// TIA Portal project "QPLC_LADDER" (V16)

(* hardware
DEVICE "S7-1200 station_1"  S7-1200 Station
   slot 0: "Rack_0"  S7-1200 Rack  Rack  V1.0
   slot 1: "PLC_1"  CPU 1214C DC/DC/DC  6ES7 214-1AG40-0XB0  V4.4
   slot 2: "DI 8/DQ 8x24VDC_1"  6ES7 223-1BH32-0XB0  V2.0
*)

// ===== PLC "PLC_1"  CPU 1214C DC/DC/DC =====

VAR_GLOBAL   // PLC tag table "Default tag table"
   "start" AT %I0.0 : Bool;   // Botão começar produção
   "stop" AT %I0.1 : Bool;   // Botão parar produção
   "reset" AT %I0.2 : Bool;   // Botão Reset produção
   "chave" AT %I0.3 : Bool;   // Seleção Modo Automático/Manual
   "Emergência (NO)" AT %I0.4 : Bool;   // Botão de emergencia NO
   "Sen_Peça_Inicial" AT %I0.5 : Bool;   // Sensor detetor de peça
   "Sensor Posição 2" AT %I0.6 : Bool;
   "Sensor Posição 3" AT %I0.7 : Bool;
   "Sen_Gripper_Embaixo" AT %I1.0 : Bool;   // Sensor do braço avançado
   "Sen_Gripper_Em_Cima" AT %I1.1 : Bool;   // Sensor do braço Recuado
   "Sen_Garra_Função" AT %I1.2 : Bool;   // Posição da garra
   "Sensor Posição 1" AT %I1.3 : Bool;   // Posição 1 do braço
   "Prato_Rec" AT %I1.4 : Bool;
   "Prato_Avanc" AT %I1.5 : Bool;
   "Btn_NC_Em" AT %I1.6 : Bool;   // Botão de emergencia NO
   "Pressostato" AT %I1.7 : Bool;
   "LedStart_KA1" AT %Q0.0 : Bool;
   "LedReset_KA2" AT %Q0.1 : Bool;
   "LedQ1_KA3" AT %Q0.2 : Bool;   // Também vai para a o sinalizador da torre
   "LEDQ2_KA4" AT %Q0.3 : Bool;
   "Braço_Direita" AT %Q0.4 : Bool;   // Ordem mover braço para esquerda
   "Braço_Esquerda" AT %Q0.5 : Bool;   // Ordem mover braço para direita
   "Braço_Ação" AT %Q0.6 : Bool;   // Ordem de avanço do braço
   "Garra_AbertaKA8" AT %Q0.7 : Bool;   // Ordem abertura da garra
   "Prato_Rec_KA9" AT %Q1.0 : Bool;   // Ordem recuar o prato
   "Prato_Avan_KA10" AT %Q1.1 : Bool;   // Ordem avançar o prato
   "Valv_KA11" AT %Q1.2 : Bool;
   "System_Byte" AT %MB1 : Byte;
   "FirstScan" AT %M1.0 : Bool;
   "DiagStatusUpdate" AT %M1.1 : Bool;
   "AlwaysTRUE" AT %M1.2 : Bool;
   "AlwaysFALSE" AT %M1.3 : Bool;
   "E_1" AT %M2.0 : Bool;
   "E_2" AT %M2.1 : Bool;
   "E_3" AT %M2.2 : Bool;
   "E_4" AT %M2.3 : Bool;
   "E_5" AT %M2.4 : Bool;
END_VAR

// folder: System blocks/Program resources

DATA_BLOCK "Cooldown para Direita"   // DB1
{ S7_Optimized_Access := 'TRUE' }
AUTHOR : Simatic
FAMILY : IEC
NAME : IEC_TMR
VERSION : 1.0
// stored: InstanceOfName IEC_TIMER
"IEC_TIMER"
BEGIN
END_DATA_BLOCK

DATA_BLOCK "Bit_ON_E2"   // DB2
{ S7_Optimized_Access := 'TRUE' }
AUTHOR : Simatic
FAMILY : IEC
NAME : IEC_TMR
VERSION : 1.0
// stored: InstanceOfName IEC_TIMER
"IEC_TIMER"
BEGIN
END_DATA_BLOCK

// folder: (top level)

FUNCTION "Geral" : Void   // FC1, LAD
{ S7_Optimized_Access := 'TRUE' }
VERSION : 0.1
BEGIN

REGION Network 1: Ordem mover braço para esquerda
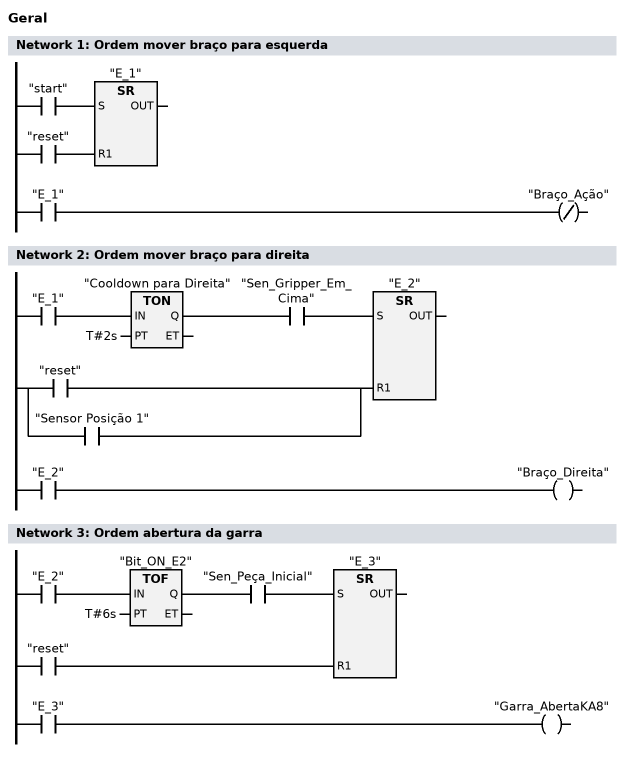
   RUNG wire#powerrail
      Contact( "start" )
      S_SR(operand := "E_1", r1 := wire#w1)
   END_RUNG
   RUNG wire#powerrail
      Contact( "reset" )
   END_RUNG wire#w1
   RUNG wire#powerrail
      Contact( "E_1" )
      I_Coil( "Braço_Ação" )
   END_RUNG
   // the same network as SCL:
   IF "start" THEN
       "E_1" := TRUE;   // SR flip-flop
   END_IF;
   IF "reset" THEN "E_1" := FALSE; END_IF;
   "Braço_Ação" := NOT "E_1";
END_REGION

REGION Network 2: Ordem mover braço para direita
   "Cooldown para Direita".TON(IN := "E_1", PT := T#2s);
   IF "Cooldown para Direita".Q AND "Sen_Gripper_Em_Cima" THEN
       "E_2" := TRUE;   // SR flip-flop
   END_IF;
   IF "reset" OR "Sensor Posição 1" THEN "E_2" := FALSE; END_IF;
   "Braço_Direita" := "E_2";
END_REGION

REGION Network 3: Ordem abertura da garra
   "Bit_ON_E2".TOF(IN := "E_2", PT := T#6s);
   IF "Bit_ON_E2".Q AND "Sen_Peça_Inicial" THEN
       "E_3" := TRUE;   // SR flip-flop
   END_IF;
   IF "reset" THEN "E_3" := FALSE; END_IF;
   "Garra_AbertaKA8" := "E_3";
END_REGION
END_FUNCTION

FUNCTION "Outputs" : Void   // FC2, LAD
{ S7_Optimized_Access := 'TRUE' }
VERSION : 0.1
BEGIN
END_FUNCTION

FUNCTION "Timers" : Void   // FC3, LAD
{ S7_Optimized_Access := 'TRUE' }
VERSION : 0.1
BEGIN
END_FUNCTION

ORGANIZATION_BLOCK "Main"   // OB1, LAD, ProgramCycle
TITLE = "Main Program Sweep (Cycle)"
{ S7_Optimized_Access := 'TRUE' }
VERSION : 0.1
// EXTRUTURA DO PROGRAMA
   VAR_INPUT
      Initial_Call : Bool;   // Initial call of this OB
      Remanence : Bool;   // =True, if remanent data are available
   END_VAR
BEGIN

REGION Network 1
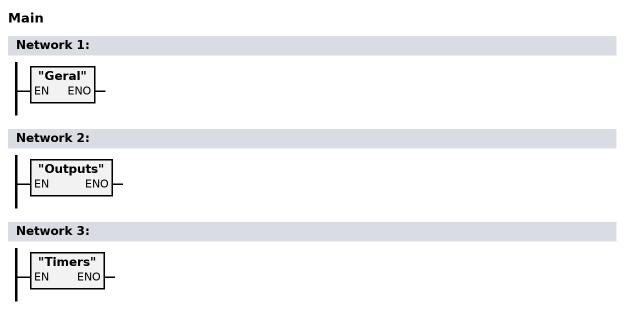
   RUNG wire#powerrail
      "Geral"()
   END_RUNG
   // the same network as SCL:
   "Geral"();
END_REGION

REGION Network 2
   RUNG wire#powerrail
      "Outputs"()
   END_RUNG
   // the same network as SCL:
   "Outputs"();
END_REGION

REGION Network 3
   RUNG wire#powerrail
      "Timers"()
   END_RUNG
   // the same network as SCL:
   "Timers"();
END_REGION
END_ORGANIZATION_BLOCK